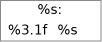
VISUALIZATION VisuAnalogChannel_Holow  // 102x42
VAR_INPUT
	Name: WSTRING;
	Unit: WSTRING;
END_VAR
VAR_IN_OUT
	fbAnalChan : FB_AnalogChannel;
END_VAR
    Rectangle (0,0 100x40), "%s:", text variable: Name, colour toggle: fbAnalChan.Error AND Tc3Sakhnenko.LibAlarm.Blink
        OnMouseDown: write fbAnalChan.Shift via Default, min 0, max 100
    Rectangle (0,20 55x20), "%3.1f", text variable: fbAnalChan.Value
    Rectangle (50,20 50x20), "%s", text variable: Unit
END_VISUALIZATION

(* stored: Version 1.1.0.1, ProductVersion 3.1.4024.2
   Visu VisuAnalogChannel_Holow: Id {90091fa4-7a82-4b88-bf7c-46b0810480c0} *)
